// TwinCAT 3 PLC project Untitled1
// ProgramVersion: 1.0.0.0
// libraries:
//   Tc2_Standard, * (Beckhoff Automation GmbH)
//   Tc2_System, * (Beckhoff Automation GmbH)
//   Tc3_Module, * (Beckhoff Automation GmbH)
// project tree:
//   / PlcTask.TcTTO
//   POUs/ DuplicateArray.TcPOU, GVL.TcGVL, Heapify.TcPOU, HeapSort.TcPOU, MAIN.TcPOU, RandomizeArray.TcPOU, SortArray.TcPOU
// real-time tasks:
//   TASK PlcTask: cycle T#10ms, priority 20, ADS port 350

CONFIGURATION Untitled1
    RESOURCE PLC ON TwinCAT3
        TASK PlcTask(INTERVAL := T#10ms, PRIORITY := 20);
        PROGRAM MAIN WITH PlcTask : MAIN;
    END_RESOURCE
END_CONFIGURATION

// ---- POUs/GVL.TcGVL
{attribute 'qualified_only'}
VAR_GLOBAL
	rand_generator: DRAND := (Seed := 154);
END_VAR

// ---- POUs/MAIN.TcPOU
PROGRAM MAIN
VAR
	unsorted : ARRAY [1..101] OF LREAL;
	unsorted2 : ARRAY [1..101] OF LREAL;
	lower: DINT;
	i: DINT;
	upper: DINT;
	rand_generator: DRAND := (Seed := 154);
END_VAR

RandomizeArray(target := unsorted);
DuplicateArray(target := unsorted2, source := unsorted);

SortArray(target := unsorted);

HeapSort(target := unsorted2);

END_PROGRAM

// ---- POUs/RandomizeArray.TcPOU
FUNCTION RandomizeArray
VAR
	lower: DINT;
	upper: DINT;
	i: DINT;

END_VAR
VAR_IN_OUT
	target: ARRAY[*] OF LREAL;
END_VAR

lower := LOWER_BOUND(target, 1);
upper := UPPER_BOUND(target, 1);

FOR i:=lower TO upper DO
  GVL.rand_generator(Num=>target[i]);
END_FOR

END_FUNCTION

// ---- POUs/DuplicateArray.TcPOU
FUNCTION DuplicateArray : INT
VAR
	lower: DINT;
	upper: DINT;
	i: DINT;
END_VAR

VAR_IN_OUT
	target: ARRAY[*] OF LREAL;
END_VAR


VAR_INPUT
	source: ARRAY[*] OF LREAL;
END_VAR

lower := LOWER_BOUND(target, 1);
upper := UPPER_BOUND(target, 1);

FOR i:=lower TO upper DO
  target[i] := source[i];
END_FOR

END_FUNCTION

// ---- POUs/SortArray.TcPOU
// Code generated by OpenAI
// Model used:	gpt-3.5-turbo
// TwinCAT Chat powered by ChatGPT:	3.6
// Time:	Monday, September 18, 2023 4:03 PM
FUNCTION SortArray
VAR
    i : DINT; 
    j : DINT; 
    temp : LREAL;
    upperbound : DINT;
	lowerbound : DINT;
END_VAR  
VAR_IN_OUT
	target: ARRAY[*] OF LREAL;
END_VAR

lowerbound := LOWER_BOUND(target, 1); 
upperbound := UPPER_BOUND(target, 1); // get array size

FOR i := lowerbound TO upperbound DO
    FOR j := lowerbound TO upperbound - i DO
        IF target[j] > target[j + 1] THEN
    // Swap the elements
            temp := target[j];
            target[j] := target[j + 1];
            target[j + 1] := temp;
        END_IF;
    END_FOR;
END_FOR;

END_FUNCTION

// ---- POUs/HeapSort.TcPOU
// Code generated by OpenAI
// Model used:	gpt-3.5-turbo
// TwinCAT Chat powered by ChatGPT:	3.6
// Time:	Monday, September 18, 2023 4:10 PM
FUNCTION HeapSort
VAR
	i : DINT;
	temp : LREAL;
	upperbound : DINT;
	lowerbound: DINT;
END_VAR
VAR_IN_OUT
	target: ARRAY[*] OF LREAL;
END_VAR

// Build heap
upperbound := UPPER_BOUND(target, 1);
lowerbound := LOWER_BOUND(target, 1);
FOR i := (upperbound + lowerbound) / 2 TO lowerbound BY -1 DO
  Heapify(upperbound, i, target);
END_FOR;

// One by one extract an element from heap
FOR i := upperbound TO (lowerbound + 1) BY -1 DO
  // Move current root to end
  temp := target[lowerbound];
  target[lowerbound] := target[i];
  target[i] := temp;

  // Call max heapify on the reduced heap
  Heapify(i, lowerbound, target);
END_FOR;

END_FUNCTION

// ---- POUs/Heapify.TcPOU
// Code generated by OpenAI
// Model used:	gpt-3.5-turbo
// TwinCAT Chat powered by ChatGPT:	3.6
// Time:	Monday, September 18, 2023 4:17 PM
FUNCTION Heapify
VAR_INPUT
	upper : DINT;
	i : DINT;
END_VAR
VAR
	largest : DINT;
	left : DINT;
	right : DINT;
	temp : LREAL;
END_VAR
VAR_IN_OUT
	target: ARRAY[*] OF LREAL;
END_VAR

// Initialize largest as root
largest := i;
left := 2 * i;
right := 2 * i + 1;

// If left child is larger than root
IF left < upper THEN 
	IF target[left] > target[largest] THEN
		largest := left;
	END_IF;
END_IF;

// If right child is larger than largest so far
IF right < upper THEN
	IF target[right] > target[largest] THEN
		largest := right;
	END_IF;
END_IF;

// If largest is not root
IF largest <> i THEN
	temp := target[i];
	target[i] := target[largest];
	target[largest] := temp;

	// Recursively heapify the affected sub-tree
	Heapify(upper, largest, target);
END_IF;

END_FUNCTION
